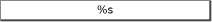
VISUALIZATION VISU_StatusWidget  // 212x22
VAR_IN_OUT
	widget : StatusWidget;
END_VAR
    Rectangle (0,0 210x20), "%s", text variable: widget.text, colour variable: widget.color.bg
        p55702900: widget.color.fg
END_VISUALIZATION

(* stored: Version 1.1.0.1, ProductVersion 3.1.0.36
   Visu VISU_StatusWidget: Id {bedae24d-8856-4e34-a079-499919c7f9e5} *)
